FUNCTION_BLOCK CU030DialogContent EXTENDS TcoCore.TcoInputDialogContentContainer
VAR_INPUT
END_VAR
VAR_OUTPUT
END_VAR
VAR
	{attribute addProperty Name "<#Recipe#>"}
	Recipe:STRING;
	{attribute addProperty Name "<#Qantity#>"}
	RequiredQuantity:INT;
	{attribute addProperty Name "<#Timeout#>"}
	Timeout:DATE_AND_TIME;
	{attribute addProperty Name "<#Exclude#>"}
	Exclude:BOOL;

END_VAR

END_FUNCTION_BLOCK

(* stored: Version 1.1.0.1
   POU CU030DialogContent: Id {f31ed13b-4691-4ea4-8777-6158a0f50d0b}, SpecialFunc None *)
